// TIA Portal V17 export
// export: Created 2023-02-13T11:16:22.0326823Z, ExportSetting WithDefaults, DisplayName Totally Integrated Automation Portal, DisplayVersion V17, DisplayName TIA Portal Openness, DisplayVersion V17, DisplayName TIA Portal Teamcenter Gateway, DisplayVersion V17, DisplayName TIA Portal Version Control Interface, DisplayVersion V17, DisplayName SINAMICS Startdrive Advanced, DisplayVersion V17, DisplayName SINAMICS Startdrive G130, G150, S120, S150, SINAMICS MV, S210, DisplayVersion V17, DisplayName SINAMICS Startdrive G110M, G120, G120C, G120D, G120P, G115D, DisplayVersion V17, DisplayName STEP 7 Professional, DisplayVersion V17, DisplayName STEP 7 Safety, DisplayVersion V17, DisplayName WinCC Professional, DisplayVersion V17
DATA_BLOCK "IO_Valve_Blend30_DB"   // DB60
VERSION : 0.1
// stored: AutoNumber true, DBAccessibleFromOPCUA true, DBAccessibleFromWebserver true, InstanceOfName IO_Valve_Blend30, InstanceOfType FB
"IO_Valve_Blend30"
   // VAR_INPUT
   //    "lock 1" : Bool;
   //    "lock 2" : Bool;
   //    "lock 3" : Bool;
   //    "lock 4" : Bool;
   //    init : Bool;
   //    reset : Bool;
   //    testing : Bool;
   // END_VAR
   // VAR
   //    "AV-30.01" : "Valve";
   //    "AV-30.02" : "Valve";
   //    "AV-30.03" : "Valve";
   //    "AV-30.04" : "Valve";
   //    "AV-30.05" : "Valve";
   //    "AV-30.06" : "Valve";
   //    "AV-30.07" : "Valve";
   //    "AV-30.08" : "Valve";
   //    "AV-30.09" : "Valve";
   //    "AV-30.10" : "Valve";
   //    "AV-30.11" : "Valve";
   //    "AV-30.12" : "Valve";
   //    "AV-30.13" : "Valve";
   //    "AV-30.14" : "Valve";
   //    "AV-30.15" : "Valve";
   //    "AV-30.16" : "Valve";
   //    "AV-30.17" : "Valve";
   //    "AV-30.18" : "Valve";
   //    "AV-30.19" : "Valve";
   //    "AV-30.20" : "Valve";
   //    "AV-30.21" : "Valve";
   //    "AV-30.22" : "Valve";
   //    "AV-30.23" : "Valve";
   //    "AV-30.24" : "Valve";
   //    "AV-30.25" : "Valve";
   //    "AV-30.26" : "Valve";
   //    "AV-30.27" : "Valve";
   //    "AV-30.28" : "Valve";
   //    "AV-30.29" : "Valve";
   //    "AV-30.30" : "Valve";
   //    "AV-30.31" : "Valve";
   //    "AV-30.32" : "Valve";
   //    "AV-30.33" : "Valve";
   //    "AV-30.34" : "Valve";
   //    "AV-30.35" : "Valve";
   //    "AV-30.36" : "Valve";
   //    "AV-30.41" : "Valve";
   //    "AV-30.42" : "Valve";
   // END_VAR
BEGIN
END_DATA_BLOCK
